FUNCTION kWToCurrent : REAL
VAR_INPUT
	kw			: REAL;
	linevoltage	: REAL;
END_VAR

IF linevoltage > 100 THEN
	kWToCurrent := kw *1000 / (linevoltage * 1.73);
ELSE
	kWToCurrent := kw *1000 / (400 * 1.73);
END_IF

END_FUNCTION

(* stored: Version 1.1.0.1, ProductVersion 3.1.4026.18
   POU kWToCurrent: Id {32729d80-6894-44ee-9769-9e7bb5830d11}, SpecialFunc None *)
